TYPE Status_KK : (Initialisieren, Lesen, Kuehlen, Abtauen, Vollautomatik, Manuell, Anlagenschutz, Schreiben);
END_TYPE

(* stored: Version 1.1.0.1, ProductVersion 3.1.4019.2
   DUT Status_KK: Id {9c78300b-74a9-4626-a375-a9a377526c19} *)
